INTERFACE I_WorkerParams

PROPERTY pCTManager : POINTER TO FB_CTManagerDefGrid
GET
END_GET
END_PROPERTY

END_INTERFACE

(* stored: Version 1.1.0.1, ProductVersion 3.1.4024.11
   Itf I_WorkerParams: Id {266da92d-f54b-43ea-b59c-0109178d5344}
   Property pCTManager: Id {b023f623-44f7-4991-83f0-5e16e98745c3}
   Get Get: Id {a4d73a7e-8965-46e2-84ae-0103fc837639} *)
